// TIA Portal V17 export
// export: Created 2024-06-16T17:47:39.8445291Z, ExportSetting WithDefaults, DisplayName Totally Integrated Automation Portal, DisplayVersion V17, DisplayName TIA Portal Openness, DisplayVersion V17, DisplayName TIA Portal Version Control Interface, DisplayVersion V17, DisplayName STEP 7 Professional, DisplayVersion V17, DisplayName STEP 7 Safety, DisplayVersion V17, DisplayName WinCC Professional, DisplayVersion V17
VAR_GLOBAL   // PLC tag table "St4_In"
   IO_Loquet_Haut AT %I4.1 : Bool;   // Loquet haut : Pas de déplacement barquette
   IO_Cpt_M AT %I4.2 : Bool;   // Présence pile en zone de marquage
   IO_PincesDC_Ouvert AT %I4.3 : Bool;   // Pinces de préhension Déchagement C : Ouverte
   IO_PincesDC_Fermee AT %I4.4 : Bool;   // Pinces de préhension Déchagement C : Fermée
   IO_Cpt_DC1 AT %I4.5 : Bool;   // Présence pile en zone Déchagement C1
   IO_Cpt_DC2 AT %I4.6 : Bool;   // Présence pile en zone Déchagement : C2
   IO_PoussoirC_Haut AT %I4.7 : Bool;   // Poussoir C en position : Haut
   IO_PincesDNC_Ouvert AT %I5.0 : Bool;   // Pinces de préhension Déchagement NC : Ouverte
   IO_PincesDNC_Fermee AT %I5.1 : Bool;   // Pinces de préhension Déchagement NC : Ferméee
   IO_Cpt_DNC0 AT %I5.2 : Bool;   // Présence pile en zone Déchagement NC0
   IO_Cpt_DNC1 AT %I5.3 : Bool;   // Présence pile en zone Déchagement DNC1
   IO_Cpt_DNC2 AT %I5.4 : Bool;   // Présence pile en zone Déchagement DNC2
   IO_PoussoirNC_Haut AT %I5.5 : Bool;   // Poussoir NC en position : Haut
END_VAR
